LIN {X 0,Y 93.556,Z 371.924,A -85,B 0,C 180,E1 -29010.244,E2 -29010.244} C_VEL
LIN {X 0,Y 85.341,Z 378.057,A -85,B 0,C 180,E1 -29014.562,E2 -29014.562} C_VEL
LIN {X 0,Y 77.823,Z 383.122,A -85,B 0,C 180,E1 -29019.86,E2 -29019.86} C_VEL
LIN {X 0,Y 71.051,Z 387.18,A -85,B 0,C 180,E1 -29026.18,E2 -29026.18} C_VEL
LIN {X 0,Y 63.393,Z 391.289,A -85,B 0,C 180,E1 -29036.337,E2 -29036.337} C_VEL
LIN {X 0,Y 58.198,Z 393.964,A -85,B 0,C 180,E1 -29048.76,E2 -29048.76} C_VEL
LIN {X 0,Y 55.707,Z 395.293,A -85,B 0,C 180,E1 -29062.753,E2 -29062.753} C_VEL
LIN {X 0,Y 55.465,Z 395.448,A -85,B 0,C 180,E1 -29070.823,E2 -29070.823} C_VEL
LIN {X 0,Y 56.614,Z 394.833,A -85,B 0,C 180,E1 -29084.376,E2 -29084.376} C_VEL
LIN {X 0,Y 60.463,Z 392.873,A -85,B 0,C 180,E1 -29097.708,E2 -29097.708} C_VEL
LIN {X 0,Y 61.587,Z 392.252,A -85,B 0,C 180,E1 -29100.259,E2 -29100.259} C_VEL
LIN {X 0,Y 63.551,Z 391.021,A -85,B 0,C 180,E1 -29105.236,E2 -29105.236} C_VEL
LIN {X 0,Y 66.186,Z 388.611,A -85,B 0,C 180,E1 -29113.429,E2 -29113.429} C_VEL
LIN {X 0,Y 68.946,Z 386.319,A -85,B 0,C 180,E1 -29119.462,E2 -29119.462} C_VEL
LIN {X 0,Y 71.966,Z 384.27,A -85,B 0,C 180,E1 -29123.268,E2 -29123.268} C_VEL
LIN {X 0,Y 73.201,Z 383.515,A -85,B 0,C 180,E1 -29124.331,E2 -29124.331} C_VEL
LIN {X 0,Y 81.467,Z 378.384,A -85,B 0,C 180,E1 -29129.621,E2 -29129.621} C_VEL
LIN {X 0,Y 91.635,Z 371.182,A -85,B 0,C 180,E1 -29134.314,E2 -29134.314} C_VEL
LIN {X 0,Y 101.567,Z 362.857,A -85,B 0,C 180,E1 -29137.943,E2 -29137.943} C_VEL
LIN {X 0,Y 102.37,Z 361.251,A -85,B 0,C 180,E1 -29139.924,E2 -29139.924} C_VEL
LIN {X 0,Y 103.137,Z 359.433,A -85,B 0,C 180,E1 -29142.555,E2 -29142.555} C_VEL
LIN {X 0,Y 103.44,Z 358.51,A -85,B 0,C 180,E1 -29144.23,E2 -29144.23} C_VEL
LIN {X 0,Y 103.685,Z 356.844,A -85,B 0,C 180,E1 -29148.267,E2 -29148.267} C_VEL
LIN {X 0,Y 104.697,Z 354.382,A -85,B 0,C 180,E1 -29156.151,E2 -29156.151} C_VEL
LIN {X 0,Y 105.195,Z 353.806,A -85,B 0,C 180,E1 -29160,E2 -29160} C_VEL
LIN {X 0,Y 104.812,Z 354.536,A -85,B 0,C 180,E1 -29163.844,E2 -29163.844} C_VEL
LIN {X 0,Y 104.278,Z 355.825,A -85,B 0,C 180,E1 -29167.746,E2 -29167.746} C_VEL
LIN {X 0,Y 103.735,Z 357.582,A -85,B 0,C 180,E1 -29171.727,E2 -29171.727} C_VEL
LIN {X 0,Y 103.406,Z 358.759,A -85,B 0,C 180,E1 -29173.906,E2 -29173.906} C_VEL
LIN {X 0,Y 102.044,Z 361.759,A -85,B 0,C 180,E1 -29178.052,E2 -29178.052} C_VEL
LIN {X 0,Y 101.123,Z 363.68,A -85,B 0,C 180,E1 -29180.334,E2 -29180.334} C_VEL
LIN {X 0,Y 100.227,Z 364.938,A -85,B 0,C 180,E1 -29181.51,E2 -29181.51} C_VEL
LIN {X 0,Y 90.999,Z 372.641,A -85,B 0,C 180,E1 -29184.841,E2 -29184.841} C_VEL
LIN {X 0,Y 80.826,Z 379.907,A -85,B 0,C 180,E1 -29189.595,E2 -29189.595} C_VEL
LIN {X 0,Y 70.127,Z 386.443,A -85,B 0,C 180,E1 -29196.702,E2 -29196.702} C_VEL
LIN {X 0,Y 60.842,Z 391.339,A -85,B 0,C 180,E1 -29206.125,E2 -29206.125} C_VEL
LIN {X 0,Y 53.548,Z 394.745,A -85,B 0,C 180,E1 -29218.331,E2 -29218.331} C_VEL
LIN {X 0,Y 49.282,Z 396.766,A -85,B 0,C 180,E1 -29233.427,E2 -29233.427} C_VEL
LIN {X 0,Y 48.314,Z 397.435,A -85,B 0,C 180,E1 -29249.999,E2 -29249.999} C_VEL
LIN {X 0,Y 49.28,Z 396.735,A -85,B 0,C 180,E1 -29266.572,E2 -29266.572} C_VEL
LIN {X 0,Y 53.544,Z 394.688,A -85,B 0,C 180,E1 -29281.669,E2 -29281.669} C_VEL
LIN {X 0,Y 60.83,Z 391.251,A -85,B 0,C 180,E1 -29293.884,E2 -29293.884} C_VEL
LIN {X 0,Y 70.132,Z 386.32,A -85,B 0,C 180,E1 -29303.291,E2 -29303.291} C_VEL
LIN {X 0,Y 80.82,Z 379.751,A -85,B 0,C 180,E1 -29310.41,E2 -29310.41} C_VEL
LIN {X 0,Y 90.994,Z 372.449,A -85,B 0,C 180,E1 -29315.165,E2 -29315.165} C_VEL
LIN {X 0,Y 100.147,Z 364.765,A -85,B 0,C 180,E1 -29318.478,E2 -29318.478} C_VEL
LIN {X 0,Y 101.069,Z 363.472,A -85,B 0,C 180,E1 -29319.655,E2 -29319.655} C_VEL
LIN {X 0,Y 102.68,Z 359.961,A -85,B 0,C 180,E1 -29324.111,E2 -29324.111} C_VEL
LIN {X 0,Y 103.323,Z 358.462,A -85,B 0,C 180,E1 -29326.273,E2 -29326.273} C_VEL
LIN {X 0,Y 103.649,Z 357.368,A -85,B 0,C 180,E1 -29328.263,E2 -29328.263} C_VEL
LIN {X 0,Y 104.163,Z 355.632,A -85,B 0,C 180,E1 -29332.245,E2 -29332.245} C_VEL
LIN {X 0,Y 104.665,Z 354.364,A -85,B 0,C 180,E1 -29336.15,E2 -29336.15} C_VEL
LIN {X 0,Y 104.989,Z 353.676,A -85,B 0,C 180,E1 -29340,E2 -29340} C_VEL
LIN {X 0,Y 104.535,Z 354.216,A -85,B 0,C 180,E1 -29343.855,E2 -29343.855} C_VEL
LIN {X 0,Y 103.977,Z 355.262,A -85,B 0,C 180,E1 -29347.77,E2 -29347.77} C_VEL
LIN {X 0,Y 103.545,Z 356.651,A -85,B 0,C 180,E1 -29351.749,E2 -29351.749} C_VEL
LIN {X 0,Y 103.098,Z 359.133,A -85,B 0,C 180,E1 -29357.378,E2 -29357.378} C_VEL
LIN {X 0,Y 102.316,Z 360.993,A -85,B 0,C 180,E1 -29360.087,E2 -29360.087} C_VEL
LIN {X 0,Y 101.548,Z 362.604,A -85,B 0,C 180,E1 -29362.093,E2 -29362.093} C_VEL
LIN {X 0,Y 91.68,Z 370.949,A -85,B 0,C 180,E1 -29365.747,E2 -29365.747} C_VEL
LIN {X 0,Y 81.509,Z 378.193,A -85,B 0,C 180,E1 -29370.432,E2 -29370.432} C_VEL
LIN {X 0,Y 73.45,Z 383.259,A -85,B 0,C 180,E1 -29375.58,E2 -29375.58} C_VEL
LIN {X 0,Y 66.103,Z 387.316,A -85,B 0,C 180,E1 -29381.907,E2 -29381.907} C_VEL
LIN {X 0,Y 57.591,Z 391.425,A -85,B 0,C 180,E1 -29392.399,E2 -29392.399} C_VEL
LIN {X 0,Y 51.637,Z 394.099,A -85,B 0,C 180,E1 -29405.902,E2 -29405.902} C_VEL
LIN {X 0,Y 48.664,Z 395.428,A -85,B 0,C 180,E1 -29421.697,E2 -29421.697} C_VEL
LIN {X 0,Y 48.386,Z 395.6,A -85,B 0,C 180,E1 -29430.001,E2 -29430.001} C_VEL
LIN {X 0,Y 49.751,Z 394.968,A -85,B 0,C 180,E1 -29446.412,E2 -29446.412} C_VEL
LIN {X 0,Y 54.255,Z 393.007,A -85,B 0,C 180,E1 -29461.209,E2 -29461.209} C_VEL
LIN {X 0,Y 61.559,Z 389.666,A -85,B 0,C 180,E1 -29473.236,E2 -29473.236} C_VEL
LIN {X 0,Y 68.405,Z 386.216,A -85,B 0,C 180,E1 -29480.406,E2 -29480.406} C_VEL
LIN {X 0,Y 73.201,Z 383.515,A -85,B 0,C 180,E1 -29484.331,E2 -29484.331} C_VEL
LIN {X 0,Y 76.744,Z 381.184,A -85,B 0,C 180,E1 -29487.483,E2 -29487.483} C_VEL
LIN {X 0,Y 81.892,Z 377.118,A -85,B 0,C 180,E1 -29492.861,E2 -29492.861} C_VEL
LIN {X 0,Y 87.439,Z 372.511,A -85,B 0,C 180,E1 -29497.444,E2 -29497.444} C_VEL
LIN {X 0,Y 91.412,Z 369.325,A -85,B 0,C 180,E1 -29499.349,E2 -29499.349} C_VEL
LIN {X 0,Y 96.612,Z 365.115,A -85,B 0,C 180,E1 -29501.031,E2 -29501.031} C_VEL
LIN {X 0,Y 97.432,Z 363.695,A -85,B 0,C 180,E1 -29503.23,E2 -29503.23} C_VEL
LIN {X 0,Y 98.107,Z 361.797,A -85,B 0,C 180,E1 -29507.589,E2 -29507.589} C_VEL
LIN {X 0,Y 98.956,Z 359.813,A -85,B 0,C 180,E1 -29513.886,E2 -29513.886} C_VEL
LIN {X 0,Y 99.969,Z 358.666,A -85,B 0,C 180,E1 -29520,E2 -29520} C_VEL
LIN {X 0,Y 99.421,Z 359.482,A -85,B 0,C 180,E1 -29524.053,E2 -29524.053} C_VEL
LIN {X 0,Y 98.744,Z 360.825,A -85,B 0,C 180,E1 -29528.183,E2 -29528.183} C_VEL
LIN {X 0,Y 98.009,Z 362.667,A -85,B 0,C 180,E1 -29532.422,E2 -29532.422} C_VEL
LIN {X 0,Y 96.271,Z 365.679,A -85,B 0,C 180,E1 -29536.978,E2 -29536.978} C_VEL
LIN {X 0,Y 95.92,Z 366.247,A -85,B 0,C 180,E1 -29537.728,E2 -29537.728} C_VEL
LIN {X 0,Y 94.568,Z 367.619,A -85,B 0,C 180,E1 -29538.639,E2 -29538.639} C_VEL
LIN {X 0,Y 83.609,Z 375.829,A -85,B 0,C 180,E1 -29542.385,E2 -29542.385} C_VEL
LIN {X 0,Y 74.584,Z 381.591,A -85,B 0,C 180,E1 -29546.468,E2 -29546.468} C_VEL
LIN {X 0,Y 64.106,Z 387.368,A -85,B 0,C 180,E1 -29553.24,E2 -29553.24} C_VEL
LIN {X 0,Y 55.908,Z 391.204,A -85,B 0,C 180,E1 -29561.039,E2 -29561.039} C_VEL
LIN {X 0,Y 47.614,Z 394.61,A -85,B 0,C 180,E1 -29573.812,E2 -29573.812} C_VEL
LIN {X 0,Y 42.508,Z 396.631,A -85,B 0,C 180,E1 -29590.689,E2 -29590.689} C_VEL
LIN {X 0,Y 41.372,Z 397.134,A -85,B 0,C 180,E1 -29600.219,E2 -29600.219} C_VEL
LIN {X 0,Y 41.202,Z 397.3,A -85,B 0,C 180,E1 -29609.999,E2 -29609.999} C_VEL
LIN {X 0,Y 41.371,Z 397.118,A -85,B 0,C 180,E1 -29619.78,E2 -29619.78} C_VEL
LIN {X 0,Y 44.616,Z 395.746,A -85,B 0,C 180,E1 -29638.2,E2 -29638.2} C_VEL
LIN {X 0,Y 51.47,Z 393.013,A -85,B 0,C 180,E1 -29653.056,E2 -29653.056} C_VEL
LIN {X 0,Y 60.832,Z 388.844,A -85,B 0,C 180,E1 -29663.97,E2 -29663.97} C_VEL
LIN {X 0,Y 71.692,Z 383.114,A -85,B 0,C 180,E1 -29671.917,E2 -29671.917} C_VEL
LIN {X 0,Y 82.071,Z 376.664,A -85,B 0,C 180,E1 -29677.006,E2 -29677.006} C_VEL
LIN {X 0,Y 92.979,Z 368.66,A -85,B 0,C 180,E1 -29680.88,E2 -29680.88} C_VEL
LIN {X 0,Y 94.56,Z 367.38,A -85,B 0,C 180,E1 -29681.374,E2 -29681.374} C_VEL
LIN {X 0,Y 95.891,Z 366.005,A -85,B 0,C 180,E1 -29682.324,E2 -29682.324} C_VEL
LIN {X 0,Y 97.163,Z 363.888,A -85,B 0,C 180,E1 -29685.336,E2 -29685.336} C_VEL
LIN {X 0,Y 97.908,Z 362.484,A -85,B 0,C 180,E1 -29687.565,E2 -29687.565} C_VEL
LIN {X 0,Y 98.963,Z 359.932,A -85,B 0,C 180,E1 -29693.842,E2 -29693.842} C_VEL
LIN {X 0,Y 99.29,Z 359.315,A -85,B 0,C 180,E1 -29695.941,E2 -29695.941} C_VEL
LIN {X 0,Y 99.759,Z 358.554,A -85,B 0,C 180,E1 -29700,E2 -29700} C_VEL
LIN {X 0,Y 98.891,Z 359.536,A -85,B 0,C 180,E1 -29705.761,E2 -29705.761} C_VEL
LIN {X 0,Y 97.981,Z 361.607,A -85,B 0,C 180,E1 -29712.427,E2 -29712.427} C_VEL
LIN {X 0,Y 97.376,Z 363.464,A -85,B 0,C 180,E1 -29716.78,E2 -29716.78} C_VEL
LIN {X 0,Y 96.595,Z 364.839,A -85,B 0,C 180,E1 -29718.943,E2 -29718.943} C_VEL
LIN {X 0,Y 90.382,Z 369.91,A -85,B 0,C 180,E1 -29721.076,E2 -29721.076} C_VEL
LIN {X 0,Y 81.139,Z 376.408,A -85,B 0,C 180,E1 -29724.568,E2 -29724.568} C_VEL
LIN {X 0,Y 70.377,Z 382.903,A -85,B 0,C 180,E1 -29730.202,E2 -29730.202} C_VEL
LIN {X 0,Y 61.578,Z 387.452,A -85,B 0,C 180,E1 -29736.974,E2 -29736.974} C_VEL
LIN {X 0,Y 52.123,Z 391.561,A -85,B 0,C 180,E1 -29747.611,E2 -29747.611} C_VEL
LIN {X 0,Y 45.222,Z 394.235,A -85,B 0,C 180,E1 -29762.211,E2 -29762.211} C_VEL
LIN {X 0,Y 41.657,Z 395.563,A -85,B 0,C 180,E1 -29780.288,E2 -29780.288} C_VEL
LIN {X 0,Y 41.303,Z 395.734,A -85,B 0,C 180,E1 -29790.001,E2 -29790.001} C_VEL
LIN {X 0,Y 42.983,Z 395.102,A -85,B 0,C 180,E1 -29809.089,E2 -29809.089} C_VEL
LIN {X 0,Y 48.308,Z 393.142,A -85,B 0,C 180,E1 -29825.588,E2 -29825.588} C_VEL
LIN {X 0,Y 56.593,Z 389.8,A -85,B 0,C 180,E1 -29838.17,E2 -29838.17} C_VEL
LIN {X 0,Y 66.761,Z 384.977,A -85,B 0,C 180,E1 -29847.372,E2 -29847.372} C_VEL
LIN {X 0,Y 75.172,Z 380.318,A -85,B 0,C 180,E1 -29852.646,E2 -29852.646} C_VEL
LIN {X 0,Y 85.689,Z 373.538,A -85,B 0,C 180,E1 -29857.325,E2 -29857.325} C_VEL
LIN {X 0,Y 91.412,Z 369.325,A -85,B 0,C 180,E1 -29859.349,E2 -29859.349} C_VEL
LIN {X 0,Y 92.905,Z 367.94,A -85,B 0,C 180,E1 -29860.453,E2 -29860.453} C_VEL
LIN {X 0,Y 93.696,Z 366.749,A -85,B 0,C 180,E1 -29862.396,E2 -29862.396} C_VEL
LIN {X 0,Y 93.718,Z 365.985,A -85,B 0,C 180,E1 -29864.768,E2 -29864.768} C_VEL
LIN {X 0,Y 93.021,Z 364.843,A -85,B 0,C 180,E1 -29872.274,E2 -29872.274} C_VEL
LIN {X 0,Y 93.724,Z 363.956,A -85,B 0,C 180,E1 -29875.699,E2 -29875.699} C_VEL
LIN {X 0,Y 94.485,Z 363.296,A -85,B 0,C 180,E1 -29880,E2 -29880} C_VEL
LIN {X 0,Y 93.8,Z 364.16,A -85,B 0,C 180,E1 -29884.297,E2 -29884.297} C_VEL
LIN {X 0,Y 92.693,Z 365.993,A -85,B 0,C 180,E1 -29889.711,E2 -29889.711} C_VEL
LIN {X 0,Y 91.566,Z 367.82,A -85,B 0,C 180,E1 -29893.312,E2 -29893.312} C_VEL
LIN {X 0,Y 90.528,Z 369.021,A -85,B 0,C 180,E1 -29894.966,E2 -29894.966} C_VEL
LIN {X 0,Y 79.566,Z 376.707,A -85,B 0,C 180,E1 -29898.276,E2 -29898.276} C_VEL
LIN {X 0,Y 68.615,Z 383.122,A -85,B 0,C 180,E1 -29902.803,E2 -29902.803} C_VEL
LIN {X 0,Y 56.913,Z 388.816,A -85,B 0,C 180,E1 -29910.184,E2 -29910.184} C_VEL
LIN {X 0,Y 46.515,Z 392.951,A -85,B 0,C 180,E1 -29920.933,E2 -29920.933} C_VEL
LIN {X 0,Y 38.47,Z 395.656,A -85,B 0,C 180,E1 -29936.764,E2 -29936.764} C_VEL
LIN {X 0,Y 34.378,Z 396.999,A -85,B 0,C 180,E1 -29958.202,E2 -29958.202} C_VEL
LIN {X 0,Y 34.094,Z 397.165,A -85,B 0,C 180,E1 -29969.999,E2 -29969.999} C_VEL
LIN {X 0,Y 34.376,Z 396.983,A -85,B 0,C 180,E1 -29981.796,E2 -29981.796} C_VEL
LIN {X 0,Y 38.468,Z 395.609,A -85,B 0,C 180,E1 -30003.235,E2 -30003.235} C_VEL
LIN {X 0,Y 46.508,Z 392.877,A -85,B 0,C 180,E1 -30019.075,E2 -30019.075} C_VEL
LIN {X 0,Y 56.911,Z 388.707,A -85,B 0,C 180,E1 -30029.818,E2 -30029.818} C_VEL
LIN {X 0,Y 68.613,Z 382.977,A -85,B 0,C 180,E1 -30037.2,E2 -30037.2} C_VEL
LIN {X 0,Y 79.555,Z 376.527,A -85,B 0,C 180,E1 -30041.744,E2 -30041.744} C_VEL
LIN {X 0,Y 90.484,Z 368.83,A -85,B 0,C 180,E1 -30045.028,E2 -30045.028} C_VEL
LIN {X 0,Y 91.498,Z 367.638,A -85,B 0,C 180,E1 -30046.678,E2 -30046.678} C_VEL
LIN {X 0,Y 92.791,Z 365.44,A -85,B 0,C 180,E1 -30051.288,E2 -30051.288} C_VEL
LIN {X 0,Y 93.695,Z 363.986,A -85,B 0,C 180,E1 -30055.699,E2 -30055.699} C_VEL
LIN {X 0,Y 94.283,Z 363.189,A -85,B 0,C 180,E1 -30060,E2 -30060} C_VEL
LIN {X 0,Y 93.591,Z 363.796,A -85,B 0,C 180,E1 -30064.307,E2 -30064.307} C_VEL
LIN {X 0,Y 92.646,Z 365.148,A -85,B 0,C 180,E1 -30069.544,E2 -30069.544} C_VEL
LIN {X 0,Y 92.043,Z 366.4,A -85,B 0,C 180,E1 -30073.243,E2 -30073.243} C_VEL
LIN {X 0,Y 91.311,Z 367.594,A -85,B 0,C 180,E1 -30075.826,E2 -30075.826} C_VEL
LIN {X 0,Y 80.035,Z 375.541,A -85,B 0,C 180,E1 -30079.271,E2 -30079.271} C_VEL
LIN {X 0,Y 67.906,Z 382.588,A -85,B 0,C 180,E1 -30084.456,E2 -30084.456} C_VEL
LIN {X 0,Y 57.567,Z 387.589,A -85,B 0,C 180,E1 -30091.287,E2 -30091.287} C_VEL
LIN {X 0,Y 47.104,Z 391.697,A -85,B 0,C 180,E1 -30101.755,E2 -30101.755} C_VEL
LIN {X 0,Y 39.064,Z 394.371,A -85,B 0,C 180,E1 -30117.336,E2 -30117.336} C_VEL
LIN {X 0,Y 34.675,Z 395.698,A -85,B 0,C 180,E1 -30138.307,E2 -30138.307} C_VEL
LIN {X 0,Y 34.214,Z 395.869,A -85,B 0,C 180,E1 -30150.001,E2 -30150.001} C_VEL
LIN {X 0,Y 36.329,Z 395.237,A -85,B 0,C 180,E1 -30172.764,E2 -30172.764} C_VEL
LIN {X 0,Y 42.724,Z 393.276,A -85,B 0,C 180,E1 -30191.148,E2 -30191.148} C_VEL
LIN {X 0,Y 52.106,Z 389.935,A -85,B 0,C 180,E1 -30204.026,E2 -30204.026} C_VEL
LIN {X 0,Y 63.199,Z 385.111,A -85,B 0,C 180,E1 -30212.829,E2 -30212.829} C_VEL
LIN {X 0,Y 72.177,Z 380.452,A -85,B 0,C 180,E1 -30217.676,E2 -30217.676} C_VEL
LIN {X 0,Y 83.209,Z 373.671,A -85,B 0,C 180,E1 -30221.843,E2 -30221.843} C_VEL
LIN {X 0,Y 91.291,Z 367.843,A -85,B 0,C 180,E1 -30224.221,E2 -30224.221} C_VEL
LIN {X 0,Y 92.141,Z 366.593,A -85,B 0,C 180,E1 -30226.772,E2 -30226.772} C_VEL
LIN {X 0,Y 93.021,Z 364.843,A -85,B 0,C 180,E1 -30232.274,E2 -30232.274} C_VEL
LIN {X 0,Y 92.859,Z 364.702,A -85,B 0,C 180,E1 -30234.673,E2 -30234.673} C_VEL
LIN {X 0,Y 91.957,Z 365.258,A -85,B 0,C 180,E1 -30237.042,E2 -30237.042} C_VEL
LIN {X 0,Y 87.698,Z 368.809,A -85,B 0,C 180,E1 -30245.14,E2 -30245.14} C_VEL
LIN {X 0,Y 86.67,Z 370.201,A -85,B 0,C 180,E1 -30249.333,E2 -30249.333} C_VEL
LIN {X 0,Y 85.959,Z 371.08,A -85,B 0,C 180,E1 -30251.15,E2 -30251.15} C_VEL
LIN {X 0,Y 75.967,Z 377.585,A -85,B 0,C 180,E1 -30253.734,E2 -30253.734} C_VEL
LIN {X 0,Y 66.17,Z 382.987,A -85,B 0,C 180,E1 -30257.077,E2 -30257.077} C_VEL
LIN {X 0,Y 53.671,Z 388.682,A -85,B 0,C 180,E1 -30263.56,E2 -30263.56} C_VEL
LIN {X 0,Y 42.185,Z 392.816,A -85,B 0,C 180,E1 -30273.59,E2 -30273.59} C_VEL
LIN {X 0,Y 32.72,Z 395.521,A -85,B 0,C 180,E1 -30289.879,E2 -30289.879} C_VEL
LIN {X 0,Y 27.435,Z 396.864,A -85,B 0,C 180,E1 -30315.156,E2 -30315.156} C_VEL
LIN {X 0,Y 27,Z 397.03,A -85,B 0,C 180,E1 -30329.999,E2 -30329.999} C_VEL
LIN {X 0,Y 29.419,Z 396.328,A -85,B 0,C 180,E1 -30358.539,E2 -30358.539} C_VEL
LIN {X 0,Y 37.055,Z 394.279,A -85,B 0,C 180,E1 -30379.345,E2 -30379.345} C_VEL
LIN {X 0,Y 47.755,Z 390.842,A -85,B 0,C 180,E1 -30392.006,E2 -30392.006} C_VEL
LIN {X 0,Y 59.823,Z 385.909,A -85,B 0,C 180,E1 -30400.024,E2 -30400.024} C_VEL
LIN {X 0,Y 72.667,Z 379.34,A -85,B 0,C 180,E1 -30405.272,E2 -30405.272} C_VEL
LIN {X 0,Y 84.274,Z 372.038,A -85,B 0,C 180,E1 -30408.488,E2 -30408.488} C_VEL
LIN {X 0,Y 85.956,Z 370.856,A -85,B 0,C 180,E1 -30408.857,E2 -30408.857} C_VEL
LIN {X 0,Y 86.547,Z 370.062,A -85,B 0,C 180,E1 -30410.654,E2 -30410.654} C_VEL
LIN {X 0,Y 87.765,Z 368.466,A -85,B 0,C 180,E1 -30415.407,E2 -30415.407} C_VEL
LIN {X 0,Y 88.596,Z 367.551,A -85,B 0,C 180,E1 -30420,E2 -30420} C_VEL
LIN {X 0,Y 87.424,Z 368.515,A -85,B 0,C 180,E1 -30425.792,E2 -30425.792} C_VEL
LIN {X 0,Y 86.266,Z 370.186,A -85,B 0,C 180,E1 -30432.143,E2 -30432.143} C_VEL
LIN {X 0,Y 76.327,Z 376.681,A -85,B 0,C 180,E1 -30434.803,E2 -30434.803} C_VEL
LIN {X 0,Y 64.603,Z 383.066,A -85,B 0,C 180,E1 -30439.049,E2 -30439.049} C_VEL
LIN {X 0,Y 54.198,Z 387.725,A -85,B 0,C 180,E1 -30444.81,E2 -30444.81} C_VEL
LIN {X 0,Y 42.69,Z 391.833,A -85,B 0,C 180,E1 -30454.6,E2 -30454.6} C_VEL
LIN {X 0,Y 33.3,Z 394.506,A -85,B 0,C 180,E1 -30470.719,E2 -30470.719} C_VEL
LIN {X 0,Y 27.749,Z 395.833,A -85,B 0,C 180,E1 -30495.33,E2 -30495.33} C_VEL
LIN {X 0,Y 27.111,Z 396.003,A -85,B 0,C 180,E1 -30510.001,E2 -30510.001} C_VEL
LIN {X 0,Y 29.901,Z 395.372,A -85,B 0,C 180,E1 -30538.042,E2 -30538.042} C_VEL
LIN {X 0,Y 37.649,Z 393.411,A -85,B 0,C 180,E1 -30558.306,E2 -30558.306} C_VEL
LIN {X 0,Y 48.266,Z 390.069,A -85,B 0,C 180,E1 -30570.89,E2 -30570.89} C_VEL
LIN {X 0,Y 60.277,Z 385.246,A -85,B 0,C 180,E1 -30578.872,E2 -30578.872} C_VEL
LIN {X 0,Y 69.782,Z 380.586,A -85,B 0,C 180,E1 -30583.096,E2 -30583.096} C_VEL
LIN {X 0,Y 81.275,Z 373.804,A -85,B 0,C 180,E1 -30586.61,E2 -30586.61} C_VEL
LIN {X 0,Y 86.269,Z 370.429,A -85,B 0,C 180,E1 -30587.851,E2 -30587.851} C_VEL
LIN {X 0,Y 87.311,Z 368.928,A -85,B 0,C 180,E1 -30593.143,E2 -30593.143} C_VEL
LIN {X 0,Y 87.845,Z 368.377,A -85,B 0,C 180,E1 -30595.411,E2 -30595.411} C_VEL
LIN {X 0,Y 88.751,Z 367.677,A -85,B 0,C 180,E1 -30600,E2 -30600} C_VEL
LIN {X 0,Y 87.698,Z 368.809,A -85,B 0,C 180,E1 -30605.14,E2 -30605.14} C_VEL
LIN {X 0,Y 86.534,Z 369.833,A -85,B 0,C 180,E1 -30606.617,E2 -30606.617} C_VEL
LIN {X 0,Y 84.101,Z 371.664,A -85,B 0,C 180,E1 -30607.781,E2 -30607.781} C_VEL
LIN {X 0,Y 80.885,Z 373.776,A -85,B 0,C 180,E1 -30608.413,E2 -30608.413} C_VEL
LIN {X 0,Y 71.697,Z 379.11,A -85,B 0,C 180,E1 -30609.092,E2 -30609.092} C_VEL
LIN {X 0,Y 70.394,Z 379.797,A -85,B 0,C 180,E1 -30609.364,E2 -30609.364} C_VEL
LIN {X 0,Y 57.775,Z 385.905,A -85,B 0,C 180,E1 -30613.304,E2 -30613.304} C_VEL
LIN {X 0,Y 44.855,Z 390.8,A -85,B 0,C 180,E1 -30619.929,E2 -30619.929} C_VEL
LIN {X 0,Y 32.861,Z 394.206,A -85,B 0,C 180,E1 -30631.183,E2 -30631.183} C_VEL
LIN {X 0,Y 23.412,Z 396.226,A -85,B 0,C 180,E1 -30653.101,E2 -30653.101} C_VEL
LIN {X 0,Y 19.894,Z 396.895,A -85,B 0,C 180,E1 -30689.998,E2 -30689.998} C_VEL
LIN {X 0,Y 23.41,Z 396.193,A -85,B 0,C 180,E1 -30726.898,E2 -30726.898} C_VEL
LIN {X 0,Y 32.857,Z 394.143,A -85,B 0,C 180,E1 -30748.823,E2 -30748.823} C_VEL
LIN {X 0,Y 44.851,Z 390.706,A -85,B 0,C 180,E1 -30760.081,E2 -30760.081} C_VEL
LIN {X 0,Y 57.774,Z 385.772,A -85,B 0,C 180,E1 -30766.696,E2 -30766.696} C_VEL
LIN {X 0,Y 71.187,Z 379.203,A -85,B 0,C 180,E1 -30770.844,E2 -30770.844} C_VEL
LIN {X 0,Y 80.472,Z 373.645,A -85,B 0,C 180,E1 -30772.829,E2 -30772.829} C_VEL
LIN {X 0,Y 81.521,Z 372.714,A -85,B 0,C 180,E1 -30775.055,E2 -30775.055} C_VEL
LIN {X 0,Y 82.663,Z 371.661,A -85,B 0,C 180,E1 -30780,E2 -30780} C_VEL
LIN {X 0,Y 81.218,Z 372.75,A -85,B 0,C 180,E1 -30786.718,E2 -30786.718} C_VEL
LIN {X 0,Y 80.111,Z 373.605,A -85,B 0,C 180,E1 -30788.431,E2 -30788.431} C_VEL
LIN {X 0,Y 68.065,Z 380.54,A -85,B 0,C 180,E1 -30791.213,E2 -30791.213} C_VEL
LIN {X 0,Y 54.836,Z 386.629,A -85,B 0,C 180,E1 -30796.009,E2 -30796.009} C_VEL
LIN {X 0,Y 45.249,Z 390.101,A -85,B 0,C 180,E1 -30801.269,E2 -30801.269} C_VEL
LIN {X 0,Y 33.351,Z 393.477,A -85,B 0,C 180,E1 -30812.554,E2 -30812.554} C_VEL
LIN {X 0,Y 23.871,Z 395.47,A -85,B 0,C 180,E1 -30833.928,E2 -30833.928} C_VEL
LIN {X 0,Y 20.017,Z 396.138,A -85,B 0,C 180,E1 -30870.002,E2 -30870.002} C_VEL
LIN {X 0,Y 23.87,Z 395.506,A -85,B 0,C 180,E1 -30906.079,E2 -30906.079} C_VEL
LIN {X 0,Y 33.328,Z 393.546,A -85,B 0,C 180,E1 -30927.515,E2 -30927.515} C_VEL
LIN {X 0,Y 45.231,Z 390.203,A -85,B 0,C 180,E1 -30938.797,E2 -30938.797} C_VEL
LIN {X 0,Y 58.09,Z 385.38,A -85,B 0,C 180,E1 -30945.441,E2 -30945.441} C_VEL
LIN {X 0,Y 68.05,Z 380.72,A -85,B 0,C 180,E1 -30948.855,E2 -30948.855} C_VEL
LIN {X 0,Y 80.22,Z 373.746,A -85,B 0,C 180,E1 -30951.643,E2 -30951.643} C_VEL
LIN {X 0,Y 81.319,Z 372.9,A -85,B 0,C 180,E1 -30953.316,E2 -30953.316} C_VEL
LIN {X 0,Y 82.782,Z 371.797,A -85,B 0,C 180,E1 -30960,E2 -30960} C_VEL
LIN {X 0,Y 81.621,Z 372.859,A -85,B 0,C 180,E1 -30964.939,E2 -30964.939} C_VEL
LIN {X 0,Y 80.582,Z 373.781,A -85,B 0,C 180,E1 -30967.161,E2 -30967.161} C_VEL
LIN {X 0,Y 70.394,Z 379.797,A -85,B 0,C 180,E1 -30969.364,E2 -30969.364} C_VEL
LIN {X 0,Y 65.179,Z 382.437,A -85,B 0,C 180,E1 -30970.179,E2 -30970.179} C_VEL
LIN {X 0,Y 52.312,Z 387.647,A -85,B 0,C 180,E1 -30970.049,E2 -30970.049} C_VEL
LIN {X 0,Y 44.803,Z 390.107,A -85,B 0,C 180,E1 -30970.558,E2 -30970.558} C_VEL
LIN {X 0,Y 41.124,Z 391.177,A -85,B 0,C 180,E1 -30971.783,E2 -30971.783} C_VEL
LIN {X 0,Y 29.801,Z 394.071,A -85,B 0,C 180,E1 -30979.38,E2 -30979.38} C_VEL
LIN {X 0,Y 18.207,Z 396.091,A -85,B 0,C 180,E1 -30999.46,E2 -30999.46} C_VEL
LIN {X 0,Y 14.16,Z 396.594,A -85,B 0,C 180,E1 -31020.239,E2 -31020.239} C_VEL
LIN {X 0,Y 12.781,Z 396.76,A -85,B 0,C 180,E1 -31049.997,E2 -31049.997} C_VEL
LIN {X 0,Y 14.159,Z 396.577,A -85,B 0,C 180,E1 -31079.757,E2 -31079.757} C_VEL
LIN {X 0,Y 23.649,Z 395.201,A -85,B 0,C 180,E1 -31113.064,E2 -31113.064} C_VEL
LIN {X 0,Y 36.283,Z 392.468,A -85,B 0,C 180,E1 -31125.574,E2 -31125.574} C_VEL
LIN {X 0,Y 49.71,Z 388.296,A -85,B 0,C 180,E1 -31131.746,E2 -31131.746} C_VEL
LIN {X 0,Y 63.459,Z 382.566,A -85,B 0,C 180,E1 -31135.361,E2 -31135.361} C_VEL
LIN {X 0,Y 73.464,Z 377.373,A -85,B 0,C 180,E1 -31137.038,E2 -31137.038} C_VEL
LIN {X 0,Y 76.073,Z 375.799,A -85,B 0,C 180,E1 -31138.57,E2 -31138.57} C_VEL
LIN {X 0,Y 76.452,Z 375.532,A -85,B 0,C 180,E1 -31140,E2 -31140} C_VEL
LIN {X 0,Y 75.842,Z 375.865,A -85,B 0,C 180,E1 -31143.027,E2 -31143.027} C_VEL
LIN {X 0,Y 73.56,Z 377.198,A -85,B 0,C 180,E1 -31144.163,E2 -31144.163} C_VEL
LIN {X 0,Y 60.008,Z 384.006,A -85,B 0,C 180,E1 -31146.726,E2 -31146.726} C_VEL
LIN {X 0,Y 46.544,Z 389.179,A -85,B 0,C 180,E1 -31151.045,E2 -31151.045} C_VEL
LIN {X 0,Y 36.533,Z 392.105,A -85,B 0,C 180,E1 -31155.877,E2 -31155.877} C_VEL
LIN {X 0,Y 24.043,Z 394.777,A -85,B 0,C 180,E1 -31168.727,E2 -31168.727} C_VEL
LIN {X 0,Y 14.478,Z 396.103,A -85,B 0,C 180,E1 -31200.962,E2 -31200.962} C_VEL
LIN {X 0,Y 12.934,Z 396.272,A -85,B 0,C 180,E1 -31230.003,E2 -31230.003} C_VEL
LIN {X 0,Y 18.592,Z 395.641,A -85,B 0,C 180,E1 -31279.118,E2 -31279.118} C_VEL
LIN {X 0,Y 30.101,Z 393.681,A -85,B 0,C 180,E1 -31299.059,E2 -31299.059} C_VEL
LIN {X 0,Y 43.17,Z 390.338,A -85,B 0,C 180,E1 -31307.64,E2 -31307.64} C_VEL
LIN {X 0,Y 56.716,Z 385.514,A -85,B 0,C 180,E1 -31312.451,E2 -31312.451} C_VEL
LIN {X 0,Y 67.04,Z 380.853,A -85,B 0,C 180,E1 -31314.827,E2 -31314.827} C_VEL
LIN {X 0,Y 74.994,Z 376.562,A -85,B 0,C 180,E1 -31316.129,E2 -31316.129} C_VEL
LIN {X 0,Y 76.147,Z 375.875,A -85,B 0,C 180,E1 -31318.035,E2 -31318.035} C_VEL
LIN {X 0,Y 76.556,Z 375.664,A -85,B 0,C 180,E1 -31320,E2 -31320} C_VEL
LIN {X 0,Y 76.18,Z 375.929,A -85,B 0,C 180,E1 -31321.433,E2 -31321.433} C_VEL
LIN {X 0,Y 73.517,Z 377.534,A -85,B 0,C 180,E1 -31322.971,E2 -31322.971} C_VEL
LIN {X 0,Y 60.004,Z 384.332,A -85,B 0,C 180,E1 -31325.392,E2 -31325.392} C_VEL
LIN {X 0,Y 46.322,Z 389.593,A -85,B 0,C 180,E1 -31329.528,E2 -31329.528} C_VEL
LIN {X 0,Y 41.124,Z 391.177,A -85,B 0,C 180,E1 -31331.783,E2 -31331.783} C_VEL
LIN {X 0,Y 35.549,Z 392.691,A -85,B 0,C 180,E1 -31333.77,E2 -31333.77} C_VEL
LIN {X 0,Y 25.841,Z 394.557,A -85,B 0,C 180,E1 -31335.11,E2 -31335.11} C_VEL
LIN {X 0,Y 17.983,Z 395.611,A -85,B 0,C 180,E1 -31336.77,E2 -31336.77} C_VEL
LIN {X 0,Y 12.306,Z 396.166,A -85,B 0,C 180,E1 -31342.894,E2 -31342.894} C_VEL
LIN {X 0,Y 10.583,Z 396.291,A -85,B 0,C 180,E1 -31347.658,E2 -31347.658} C_VEL
LIN {X 0,Y 5.681,Z 396.626,A -85,B 0,C 180,E1 -31409.993,E2 -31409.993} C_VEL
LIN {X 0,Y 14.734,Z 395.921,A -85,B 0,C 180,E1 -31482.541,E2 -31482.541} C_VEL
LIN {X 0,Y 28.247,Z 393.872,A -85,B 0,C 180,E1 -31494.394,E2 -31494.394} C_VEL
LIN {X 0,Y 42.179,Z 390.433,A -85,B 0,C 180,E1 -31498.636,E2 -31498.636} C_VEL
LIN {X 0,Y 49.195,Z 388.16,A -85,B 0,C 180,E1 -31500.001,E2 -31500.001} C_VEL
LIN {X 0,Y 49.213,Z 388.135,A -85,B 0,C 180,E1 -31501.514,E2 -31501.514} C_VEL
LIN {X 0,Y 35.257,Z 392.241,A -85,B 0,C 180,E1 -31504.686,E2 -31504.686} C_VEL
LIN {X 0,Y 21.542,Z 394.913,A -85,B 0,C 180,E1 -31511.842,E2 -31511.842} C_VEL
LIN {X 0,Y 8.955,Z 396.238,A -85,B 0,C 180,E1 -31538.306,E2 -31538.306} C_VEL
LIN {X 0,Y 5.839,Z 396.407,A -85,B 0,C 180,E1 -31590.007,E2 -31590.007} C_VEL
LIN {X 0,Y 14.938,Z 395.776,A -85,B 0,C 180,E1 -31660.222,E2 -31660.222} C_VEL
LIN {X 0,Y 28.345,Z 393.816,A -85,B 0,C 180,E1 -31672.663,E2 -31672.663} C_VEL
LIN {X 0,Y 42.222,Z 390.472,A -85,B 0,C 180,E1 -31677.115,E2 -31677.115} C_VEL
LIN {X 0,Y 49.212,Z 388.254,A -85,B 0,C 180,E1 -31678.583,E2 -31678.583} C_VEL
LIN {X 0,Y 49.197,Z 388.277,A -85,B 0,C 180,E1 -31679.999,E2 -31679.999} C_VEL
LIN {X 0,Y 35.192,Z 392.412,A -85,B 0,C 180,E1 -31683.102,E2 -31683.102} C_VEL
LIN {X 0,Y 21.384,Z 395.115,A -85,B 0,C 180,E1 -31689.603,E2 -31689.603} C_VEL
LIN {X 0,Y 10.583,Z 396.291,A -85,B 0,C 180,E1 -31707.658,E2 -31707.658} C_VEL
LIN {X 0,Y 9.094,Z 398.286,A -85,B 0,C 180,E1 -31714.156,E2 -31714.156} C_VEL
LIN {X 0,Y 9.094,Z 600,A -85,B 0,C 180,E1 -31714.156,E2 -31714.156} C_VEL
LIN {X 0,Y 9.094,Z 600,A -85,B 0,C 180,E1 -31714.156,E2 -31714.156}

QRS_NEXT_CUT()

QRS_NEXT()
QRS_HOME()

END
